// SIMATIC STEP 7 (V5.x) project Q3
// CPU: CPU 313C
// station: Hardware
// station: SIMATIC 300(1)
// station: P_ADR_BUS
// program: S7 Program(1)

SYMBOL_TABLE
"Counter"	C 0	COUNTER
"Start"	I 0.0	BOOL
"Stop"	I 0.1	BOOL
"Start/Stop Mem"	M 0.0	BOOL
"Pos Trig"	M 0.1	BOOL
"Counter num"	MW 1	WORD
"Green 2"	Q 0.0	BOOL
"Yellow 2"	Q 0.1	BOOL
"Red 2"	Q 0.2	BOOL
"Green 1"	Q 0.3	BOOL
"Yellow 1"	Q 0.4	BOOL
"Red 1"	Q 0.5	BOOL
"Start button light"	Q 0.6	BOOL
"Stop button light"	Q 0.7	BOOL
"20s-Timer-1"	T 0	TIMER
"7s-Timer"	T 1	TIMER
"20s-Timer-2"	T 2	TIMER
END_SYMBOL_TABLE

ORGANIZATION_BLOCK OB 1
TITLE = "Main Program Sweep (Cycle)"
VERSION : 0.1
VAR_TEMP
  OB1_EV_CLASS : BYTE ;	//Bits 0-3 = 1 (Coming event), Bits 4-7 = 1 (Event class 1)
  OB1_SCAN_1 : BYTE ;	//1 (Cold restart scan 1 of OB 1), 3 (Scan 2-n of OB 1)
  OB1_PRIORITY : BYTE ;	//Priority of OB Execution
  OB1_OB_NUMBR : BYTE ;	//1 (Organization block 1, OB1)
  OB1_RESERVED_1 : BYTE ;	//Reserved for system
  OB1_RESERVED_2 : BYTE ;	//Reserved for system
  OB1_PREV_CYCLE : INT ;	//Cycle time of previous OB1 scan (milliseconds)
  OB1_MIN_CYCLE : INT ;	//Minimum cycle time of OB1 (milliseconds)
  OB1_MAX_CYCLE : INT ;	//Maximum cycle time of OB1 (milliseconds)
  OB1_DATE_TIME : DATE_AND_TIME ;	//Date and time OB1 started
END_VAR
BEGIN
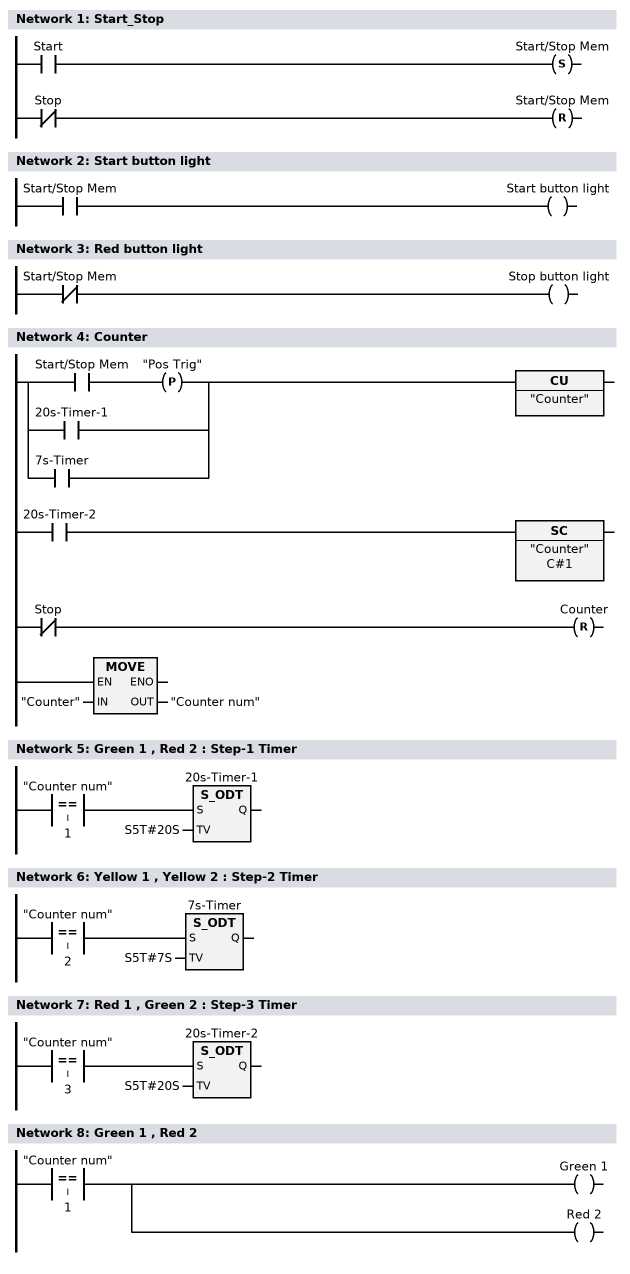
NETWORK
TITLE = Start_Stop
      A     "Start";
      S     "Start/Stop Mem";
      AN    "Stop";
      R     "Start/Stop Mem";
      NOP   0;
NETWORK
TITLE = Start button light
      A     "Start/Stop Mem";
      =     "Start button light";
NETWORK
TITLE = Red button light
      AN    "Start/Stop Mem";
      =     "Stop button light";
NETWORK
TITLE = Counter
      A(;
      O(;
      A     "Start/Stop Mem";
      BLD   100;
      FP    "Pos Trig";
      );
      O     "20s-Timer-1";
      O     "7s-Timer";
      );
      CU    "Counter";
      BLD   101;
      A     "20s-Timer-2";
      L     C#1;
      S     "Counter";
      AN    "Stop";
      R     "Counter";
      L     "Counter";
      T     "Counter num";
      NOP   0;
      NOP   0;
NETWORK
TITLE = Green 1 , Red 2 : Step-1 Timer
      A(;
      L     "Counter num";
      L     1;
      ==I;
      );
      L     S5T#20S;
      SD    "20s-Timer-1";
      NOP   0;
      NOP   0;
      NOP   0;
      NOP   0;
NETWORK
TITLE = Yellow 1 , Yellow 2 : Step-2 Timer
      A(;
      L     "Counter num";
      L     2;
      ==I;
      );
      L     S5T#7S;
      SD    "7s-Timer";
      NOP   0;
      NOP   0;
      NOP   0;
      NOP   0;
NETWORK
TITLE = Red 1 , Green 2 : Step-3 Timer
      A(;
      L     "Counter num";
      L     3;
      ==I;
      );
      L     S5T#20S;
      SD    "20s-Timer-2";
      NOP   0;
      NOP   0;
      NOP   0;
      NOP   0;
NETWORK
TITLE = Green 1 , Red 2
      L     "Counter num";
      L     1;
      ==I;
      =     "Green 1";
      =     "Red 2";
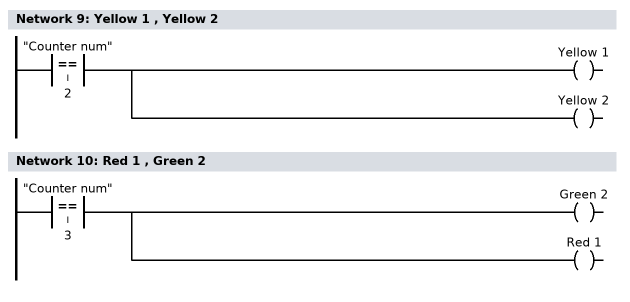
NETWORK
TITLE = Yellow 1 , Yellow 2
      L     "Counter num";
      L     2;
      ==I;
      =     "Yellow 1";
      =     "Yellow 2";
NETWORK
TITLE = Red 1 , Green 2
      L     "Counter num";
      L     3;
      ==I;
      =     "Green 2";
      =     "Red 1";
END_ORGANIZATION_BLOCK
